PROGRAM PRG_IO_Scaling
VAR
	AI1: FB_Scale;
	AI2: FB_Scale;
	AI3: FB_Scale;
	AI4: FB_Scale;
	AI5: FB_Scale;
	AI6: FB_Scale;
	AI7: FB_Scale;
	AI8: FB_Scale;
	AO1: FB_Scale;
	AO2: FB_Scale;
	AO3: FB_Scale;
	AO4: FB_Scale;
	AO5: FB_Scale;
	AO6: FB_Scale;
	AO7: FB_Scale;
	AO8: FB_Scale;
END_VAR

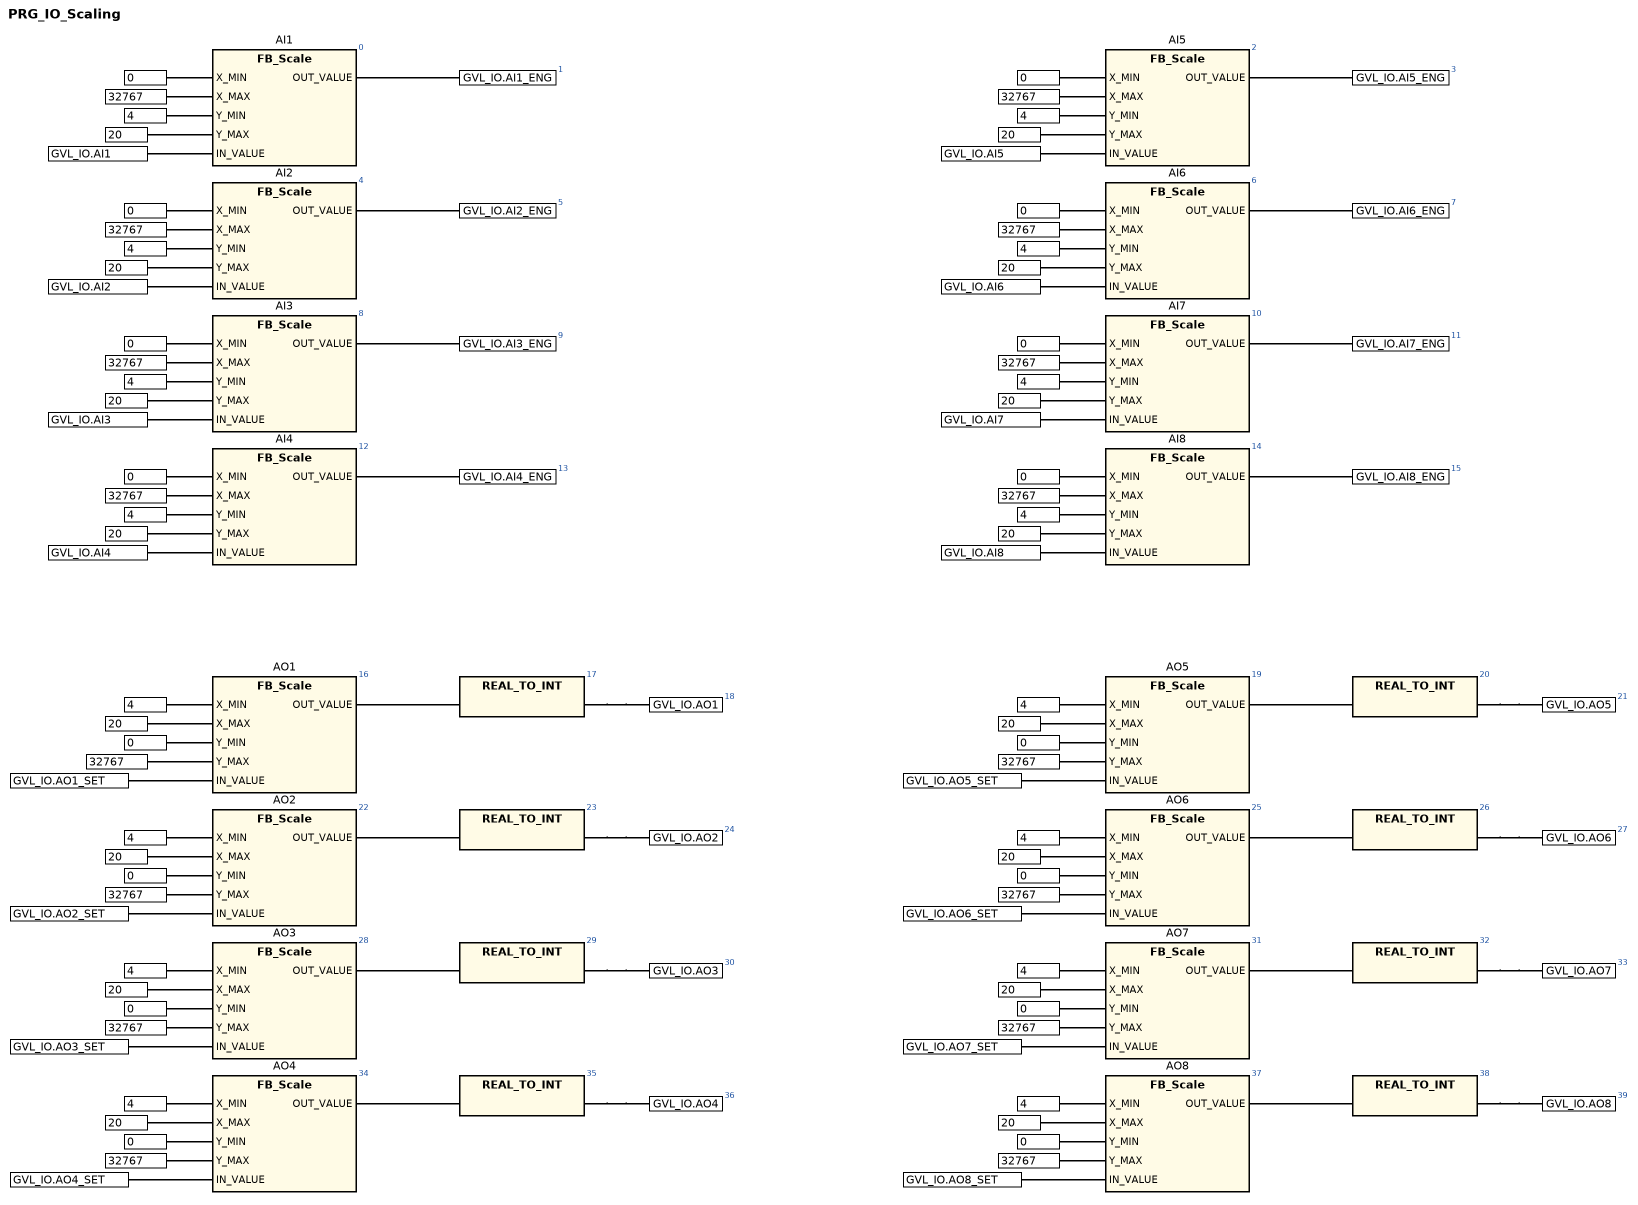
AI1(X_MIN := 0, X_MAX := 32767, Y_MIN := 4, Y_MAX := 20, IN_VALUE := GVL_IO.AI1); // FB_Scale
GVL_IO.AI1_ENG := AI1.OUT_VALUE;
AI5(X_MIN := 0, X_MAX := 32767, Y_MIN := 4, Y_MAX := 20, IN_VALUE := GVL_IO.AI5); // FB_Scale
GVL_IO.AI5_ENG := AI5.OUT_VALUE;
AI2(X_MIN := 0, X_MAX := 32767, Y_MIN := 4, Y_MAX := 20, IN_VALUE := GVL_IO.AI2); // FB_Scale
GVL_IO.AI2_ENG := AI2.OUT_VALUE;
AI6(X_MIN := 0, X_MAX := 32767, Y_MIN := 4, Y_MAX := 20, IN_VALUE := GVL_IO.AI6); // FB_Scale
GVL_IO.AI6_ENG := AI6.OUT_VALUE;
AI3(X_MIN := 0, X_MAX := 32767, Y_MIN := 4, Y_MAX := 20, IN_VALUE := GVL_IO.AI3); // FB_Scale
GVL_IO.AI3_ENG := AI3.OUT_VALUE;
AI7(X_MIN := 0, X_MAX := 32767, Y_MIN := 4, Y_MAX := 20, IN_VALUE := GVL_IO.AI7); // FB_Scale
GVL_IO.AI7_ENG := AI7.OUT_VALUE;
AI4(X_MIN := 0, X_MAX := 32767, Y_MIN := 4, Y_MAX := 20, IN_VALUE := GVL_IO.AI4); // FB_Scale
GVL_IO.AI4_ENG := AI4.OUT_VALUE;
AI8(X_MIN := 0, X_MAX := 32767, Y_MIN := 4, Y_MAX := 20, IN_VALUE := GVL_IO.AI8); // FB_Scale
GVL_IO.AI8_ENG := AI8.OUT_VALUE;
AO1(X_MIN := 4, X_MAX := 20, Y_MIN := 0, Y_MAX := 32767, IN_VALUE := GVL_IO.AO1_SET); // FB_Scale
GVL_IO.AO1 := REAL_TO_INT(AO1.OUT_VALUE);
AO5(X_MIN := 4, X_MAX := 20, Y_MIN := 0, Y_MAX := 32767, IN_VALUE := GVL_IO.AO5_SET); // FB_Scale
GVL_IO.AO5 := REAL_TO_INT(AO5.OUT_VALUE);
AO2(X_MIN := 4, X_MAX := 20, Y_MIN := 0, Y_MAX := 32767, IN_VALUE := GVL_IO.AO2_SET); // FB_Scale
GVL_IO.AO2 := REAL_TO_INT(AO2.OUT_VALUE);
AO6(X_MIN := 4, X_MAX := 20, Y_MIN := 0, Y_MAX := 32767, IN_VALUE := GVL_IO.AO6_SET); // FB_Scale
GVL_IO.AO6 := REAL_TO_INT(AO6.OUT_VALUE);
AO3(X_MIN := 4, X_MAX := 20, Y_MIN := 0, Y_MAX := 32767, IN_VALUE := GVL_IO.AO3_SET); // FB_Scale
GVL_IO.AO3 := REAL_TO_INT(AO3.OUT_VALUE);
AO7(X_MIN := 4, X_MAX := 20, Y_MIN := 0, Y_MAX := 32767, IN_VALUE := GVL_IO.AO7_SET); // FB_Scale
GVL_IO.AO7 := REAL_TO_INT(AO7.OUT_VALUE);
AO4(X_MIN := 4, X_MAX := 20, Y_MIN := 0, Y_MAX := 32767, IN_VALUE := GVL_IO.AO4_SET); // FB_Scale
GVL_IO.AO4 := REAL_TO_INT(AO4.OUT_VALUE);
AO8(X_MIN := 4, X_MAX := 20, Y_MIN := 0, Y_MAX := 32767, IN_VALUE := GVL_IO.AO8_SET); // FB_Scale
GVL_IO.AO8 := REAL_TO_INT(AO8.OUT_VALUE);

END_PROGRAM

(* stored: Version 1.1.0.1, ProductVersion 3.1.4024.4
   POU PRG_IO_Scaling: Id {59e30c98-fb2d-41a8-9b19-dfda3dc82e3e}, SpecialFunc None *)
